Staubli VAL3: goToPoint.pgx

public program goToPoint(num x_nIndexTool)
begin
  resetMotion()
  if x_nIndexTool==0
    movej(saveData:rif2,saveData:tData[x_nIndexTool].tcp,{25,25,25,9999,9999,off,50,50})
  else
    pPoint.trsf=position(saveData:rif2,world)
    pPoint.config={sfree,efree,wfree}
    movej(pPoint,saveData:tData[x_nIndexTool].tcp,{25,25,25,9999,9999,off,50,50})
  endIf
end
